(*
Interface for single-input single-output controller toolbox components.

Implementors expose a writable :attr:`Input` and a read-only :attr:`Output`,
both as ``LREAL``.
*)
INTERFACE I_SisoComponent EXTENDS I_Component

// Gets or sets the input to the component.
PROPERTY Input : LREAL
GET
END_GET
SET
END_SET
END_PROPERTY

// Gets the output produced by the component.
PROPERTY Output : LREAL
GET
END_GET
END_PROPERTY

END_INTERFACE

(* stored: Version 1.1.0.1, ProductVersion 3.1.4024.15
   Itf I_SisoComponent: Id {d0d754b4-b7d2-49a1-a76f-119a720a55c4}
   Property Input: Id {fac8086d-d94f-49ff-a29b-0b3804080a5a}
   Get Get: Id {bca0112e-91fe-44bf-8e4d-8d6bdaa62a5d}
   Set Set: Id {9b173d64-a041-4dde-aba8-0314bc3d68e1}
   Property Output: Id {02280395-c00c-4c0c-afde-7315f14eecbf}
   Get Get: Id {7b20950d-35ea-4524-8277-0c813fee378f} *)
